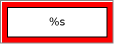
VISUALIZATION Visu_StanMaszyny_AktualyStan_BezNaciskania  // 114x44
VAR_IN_OUT
	
END_VAR
VAR_INPUT
	stVisuStan								: DUT_StanMaszyny_VISU_Stan;
END_VAR
    RoundedRectangle (2,2 110x40), invisible if: not stVisuStan.bAktywny
    RoundedRectangle (7,7 100x30), "%s", text variable: stVisuStan.sNazwa, colour variable: 16#FF000000 OR (16#FF000000 OR (stVisuStan.dwKolorTla))
END_VISUALIZATION

(* stored: Version 1.1.0.1, ProductVersion 3.1.4024.11
   Visu Visu_StanMaszyny_AktualyStan_BezNaciskania: Id {d2fe3c20-d163-4349-9420-c08a28bc1098} *)
